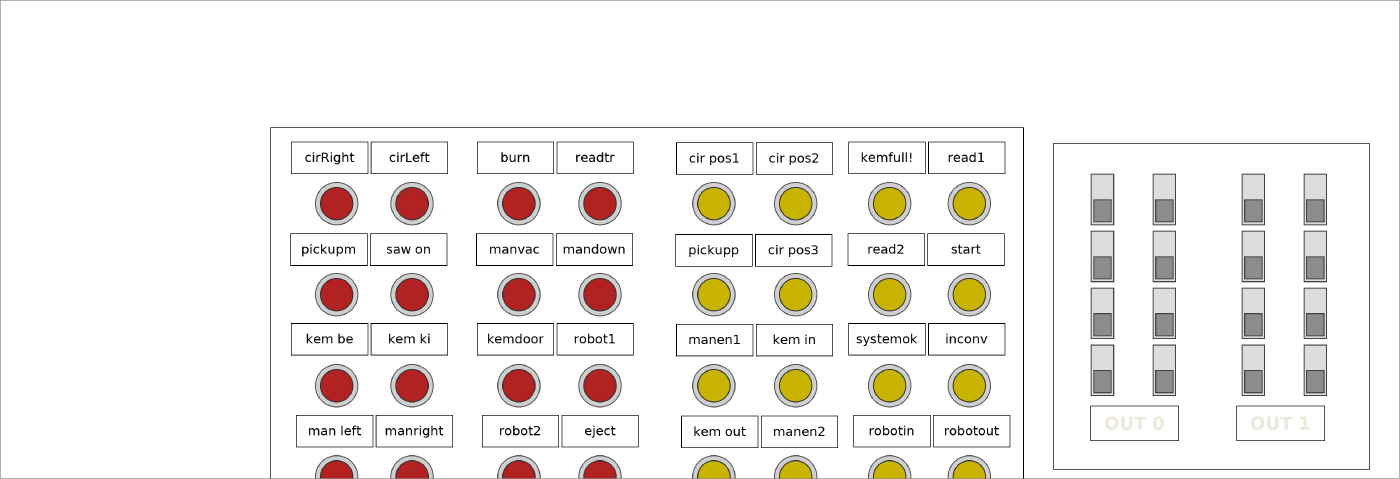
VISUALIZATION StandardPLCversenyVISU  // 1967x673
    Rectangle (1769,708 331x259)
    Rectangle (1480,201 444x459)
    Rectangle (380,179 1058x846)
    Lamp1 (438,251 70x70), variable: GIOL.out0, style: Lamp-Lamp1-Red
    Lamp1 (544,251 70x70), variable: GIOL.out1, style: Lamp-Lamp1-Red
    Lamp1 (694,251 70x70), variable: GIOL.out8, style: Lamp-Lamp1-Red
    Lamp1 (808,251 70x70), variable: GIOL.out9, style: Lamp-Lamp1-Red
    Lamp1 (438,379 70x70), variable: GIOL.out2, style: Lamp-Lamp1-Red
    Lamp1 (544,379 70x70), variable: GIOL.out3, style: Lamp-Lamp1-Red
    Lamp1 (694,379 70x70), variable: GIOL.out10, style: Lamp-Lamp1-Red
    Lamp1 (808,379 70x70), variable: GIOL.out11, style: Lamp-Lamp1-Red
    Lamp1 (438,507 70x70), variable: GIOL.out4, style: Lamp-Lamp1-Red
    Lamp1 (544,507 70x70), variable: GIOL.out5, style: Lamp-Lamp1-Red
    Lamp1 (694,507 70x70), variable: GIOL.out12, style: Lamp-Lamp1-Red
    Lamp1 (808,507 70x70), variable: GIOL.out13, style: Lamp-Lamp1-Red
    Lamp1 (438,635 70x70), variable: GIOL.out6, style: Lamp-Lamp1-Red
    Lamp1 (544,635 70x70), variable: GIOL.out7, style: Lamp-Lamp1-Red
    Lamp1 (694,635 70x70), variable: GIOL.out14, style: Lamp-Lamp1-Red
    Lamp1 (808,635 70x70), variable: GIOL.out15, style: Lamp-Lamp1-Red
    Lamp1 (968,251 70x70), variable: GIOL.in0, style: Lamp-Lamp1-Yellow
    Lamp1 (1083,251 70x70), variable: GIOL.in1, style: Lamp-Lamp1-Yellow
    Lamp1 (1215,251 70x70), variable: GIOL.in8, style: Lamp-Lamp1-Yellow
    Lamp1 (1327,251 70x70), variable: GIOL.in9, style: Lamp-Lamp1-Yellow
    Lamp1 (968,379 70x70), variable: GIOL.in2, style: Lamp-Lamp1-Yellow
    Lamp1 (1083,379 70x70), variable: GIOL.in3, style: Lamp-Lamp1-Yellow
    Lamp1 (1215,379 70x70), variable: GIOL.in10, style: Lamp-Lamp1-Yellow
    Lamp1 (1327,379 70x70), variable: GIOL.in11, style: Lamp-Lamp1-Yellow
    Lamp1 (968,507 70x70), variable: GIOL.in4, style: Lamp-Lamp1-Yellow
    Lamp1 (1083,507 70x70), variable: GIOL.in5, style: Lamp-Lamp1-Yellow
    Lamp1 (1215,507 70x70), variable: GIOL.in12, style: Lamp-Lamp1-Yellow
    Lamp1 (1327,507 70x70), variable: GIOL.in13, style: Lamp-Lamp1-Yellow
    Lamp1 (968,635 70x70), variable: GIOL.in6, style: Lamp-Lamp1-Yellow
    Lamp1 (1083,635 70x70), variable: GIOL.in7, style: Lamp-Lamp1-Yellow
    Lamp1 (1215,635 70x70), variable: GIOL.in14, style: Lamp-Lamp1-Yellow
    Lamp1 (1327,635 70x70), variable: GIOL.in15, style: Lamp-Lamp1-Yellow
    Rectangle (700,733 124x49), "OUT 1"
    Rectangle (988,728 124x49), "IN 0"
    Rectangle (450,733 124x49), "OUT 0"
    Rectangle (1229,726 124x49), "IN 1"
    Rectangle (505,888 695x68), "EXECUTING: %s", text variable: GIOL.TaskName
    DipSwitch (1600,240 72x80), variable: GIOL.out1, behaviour: TOGGLE, style: Switch-DipSwitch-Gray
    DipSwitch (1513,240 72x80), variable: GIOL.out0, behaviour: TOGGLE, style: Switch-DipSwitch-Gray
    DipSwitch (1600,320 72x80), variable: GIOL.out3, behaviour: TOGGLE, style: Switch-DipSwitch-Gray
    DipSwitch (1513,320 72x80), variable: GIOL.out2, behaviour: TOGGLE, style: Switch-DipSwitch-Gray
    DipSwitch (1600,400 72x80), variable: GIOL.out5, behaviour: TOGGLE, style: Switch-DipSwitch-Gray
    DipSwitch (1513,400 72x80), variable: GIOL.out4, behaviour: TOGGLE, style: Switch-DipSwitch-Gray
    DipSwitch (1600,480 72x80), variable: GIOL.out7, behaviour: TOGGLE, style: Switch-DipSwitch-Gray
    DipSwitch (1513,480 72x80), variable: GIOL.out6, behaviour: TOGGLE, style: Switch-DipSwitch-Gray
    DipSwitch (1812,240 72x80), variable: GIOL.out9, behaviour: TOGGLE, style: Switch-DipSwitch-Gray
    DipSwitch (1725,240 72x80), variable: GIOL.out8, behaviour: TOGGLE, style: Switch-DipSwitch-Gray
    DipSwitch (1812,320 72x80), variable: GIOL.out11, behaviour: TOGGLE, style: Switch-DipSwitch-Gray
    DipSwitch (1725,320 72x80), variable: GIOL.out10, behaviour: TOGGLE, style: Switch-DipSwitch-Gray
    DipSwitch (1812,400 72x80), variable: GIOL.out13, behaviour: TOGGLE, style: Switch-DipSwitch-Gray
    DipSwitch (1725,400 72x80), variable: GIOL.out12, behaviour: TOGGLE, style: Switch-DipSwitch-Gray
    DipSwitch (1812,480 72x80), variable: GIOL.out15, behaviour: TOGGLE, style: Switch-DipSwitch-Gray
    DipSwitch (1725,480 72x80), variable: GIOL.out14, behaviour: TOGGLE, style: Switch-DipSwitch-Gray
    Rectangle (1737,570 124x49), "OUT 1"
    Rectangle (1532,570 124x49), "OUT 0"
    Rectangle (1970,201 444x459)
    DipSwitch (2093,240 72x80), variable: GIOL.bIn1, behaviour: TOGGLE, style: Switch-DipSwitch-Gray
    DipSwitch (2006,240 72x80), variable: GIOL.bIn0, behaviour: TOGGLE, style: Switch-DipSwitch-Gray
    DipSwitch (2093,320 72x80), variable: GIOL.bIn3, behaviour: TOGGLE, style: Switch-DipSwitch-Gray
    DipSwitch (2006,320 72x80), variable: GIOL.bIn2, behaviour: TOGGLE, style: Switch-DipSwitch-Gray
    DipSwitch (2093,400 72x80), variable: GIOL.bIn5, behaviour: TOGGLE, style: Switch-DipSwitch-Gray
    DipSwitch (2006,400 72x80), variable: GIOL.bIn4, behaviour: TOGGLE, style: Switch-DipSwitch-Gray
    DipSwitch (2093,480 72x80), variable: GIOL.bIn7, behaviour: TOGGLE, style: Switch-DipSwitch-Gray
    DipSwitch (2006,480 72x80), variable: GIOL.bIn6, behaviour: TOGGLE, style: Switch-DipSwitch-Gray
    DipSwitch (2305,240 72x80), variable: GIOL.bIn9, behaviour: TOGGLE, style: Switch-DipSwitch-Gray
    DipSwitch (2218,240 72x80), variable: GIOL.bIn8, behaviour: TOGGLE, style: Switch-DipSwitch-Gray
    DipSwitch (2305,320 72x80), variable: GIOL.bIn11, behaviour: TOGGLE, style: Switch-DipSwitch-Gray
    DipSwitch (2218,320 72x80), variable: GIOL.bIn10, behaviour: TOGGLE, style: Switch-DipSwitch-Gray
    DipSwitch (2305,400 72x80), variable: GIOL.bIn13, behaviour: TOGGLE, style: Switch-DipSwitch-Gray
    DipSwitch (2218,400 72x80), variable: GIOL.bIn12, behaviour: TOGGLE, style: Switch-DipSwitch-Gray
    DipSwitch (2305,480 72x80), variable: GIOL.bIn15, behaviour: TOGGLE, style: Switch-DipSwitch-Gray
    DipSwitch (2218,480 72x80), variable: GIOL.bIn14, behaviour: TOGGLE, style: Switch-DipSwitch-Gray
    Rectangle (2230,570 124x49), "IN 1"
    Rectangle (2025,570 124x49), "IN 0"
    Rectangle (1210,888 153x68), "CASE: %d", text variable: GIOL.CaseNum
    DipSwitch (1818,753 116x113), variable: MAIN.INMODE.INState, behaviour: TOGGLE, style: Switch-DipSwitch-Gray
    Rectangle (1828,898 226x49), "INPUT MODE"
    Lamp1 (1963,775 70x70), variable: MAIN.INMODE.INState, style: Lamp-Lamp1-Yellow
    Rectangle (409,199 108x45), "cirRight"
    Rectangle (521,199 108x45), "cirLeft"
    Rectangle (670,199 108x45), "burn"
    Rectangle (782,199 108x45), "readtr"
    Rectangle (950,200 108x45), "cir pos1"
    Rectangle (1062,200 108x45), "cir pos2"
    Rectangle (1192,199 108x45), "kemfull!"
    Rectangle (1304,199 108x45), "read1"
    Rectangle (408,328 108x45), "pickupm"
    Rectangle (520,328 108x45), "saw on"
    Rectangle (669,328 108x45), "manvac"
    Rectangle (781,328 108x45), "mandown"
    Rectangle (949,329 108x45), "pickupp"
    Rectangle (1061,329 108x45), "cir pos3"
    Rectangle (1191,328 108x45), "read2"
    Rectangle (1303,328 108x45), "start"
    Rectangle (409,454 108x45), "kem be"
    Rectangle (521,454 108x45), "kem ki"
    Rectangle (670,454 108x45), "kemdoor"
    Rectangle (782,454 108x45), "robot1"
    Rectangle (950,455 108x45), "manen1"
    Rectangle (1062,455 108x45), "kem in"
    Rectangle (1192,454 108x45), "systemok"
    Rectangle (1304,454 108x45), "inconv"
    Rectangle (416,583 108x45), "man left"
    Rectangle (528,583 108x45), "manright"
    Rectangle (677,583 108x45), "robot2"
    Rectangle (789,583 108x45), "eject"
    Rectangle (957,584 108x45), "kem out"
    Rectangle (1069,584 108x45), "manen2"
    Rectangle (1199,583 108x45), "robotin"
    Rectangle (1311,583 108x45), "robotout"
END_VISUALIZATION

(* stored: Version 1.1.0.1, ProductVersion 3.1.4024.15
   Visu StandardPLCversenyVISU: Id {a8bc012b-8952-461b-92ed-7c0d35e309be} *)
